Staubli VAL3: cycleStatus.pjx

--- cycleStatus.pjx ---
Parameters version=s7.5 stackSize=5000 millimeterUnit=true
Program file=addAction.pgx
Program file=addActionTime.pgx
Program file=addTraj.pgx
Program file=checkTollerance.pgx
Program file=getAction.pgx
Program file=getLastId.pgx
Program file=getSizeAction.pgx
Program file=getTraj.pgx
Program file=init.pgx
Program file=init_logAction.pgx
Program file=isActionEmpty.pgx
Program file=printLog.pgx
Program file=putInstr_Traj.pgx
Program file=recordPowerDown.pgx
Program file=removeAction.pgx
Program file=removeAllInstr.pgx
Program file=removeTraj.pgx
Data file=cycleStatus.dtx
Library alias=tcp path=Disk://kernel/tool/tool.pjx
Library alias=saveData path=Disk://saveData/saveData.pjx
Type name=TrajectoryItem path=Disk://kernel/template/TrajectoryItem/TrajectoryItem.pjx
Type name=ActionItem path=Disk://kernel/template/ActionItem/ActionItem.pjx
Type name=InstrItem path=Disk://kernel/template/InstrItem/InstrItem.pjx
Type name=progItem path=Disk://kernel/template/progItem/progItem.pjx
Type name=Trajectory path=Disk://kernel/template/Trajectory/Trajectory.pjx

--- cycleStatus.dtx ---
public ActionItem aActionTime
  [0]
    num nDistance = 1
    num nMoveId = 3
    num nTimeId
    num nPointId
    InstrItem iInstr[3]
      [0]
        string sType
        string sData
      [1]
        string sType
        string sData
      [2]
        string sType
        string sData
    string sIdTraj = "POINT place"
public InstrItem iToSuperV
  [0]
    string sType = "PROG"
    string sData = "home"
InstrItem tcpInstr[3]
  [0]
    string sType = "OUT"
    string sData = "bOut0>ON"
  [1]
    string sType = "OUT"
    string sData = "bOut1>OFF"
  [2]
    string sType
    string sData
Trajectory tTrajCycle
  [0]
    TrajectoryItem tSuper[3]
      [0]
        num distance
        num moveType = 1
        num nTime
        num nStop
        num nTcpAction
        string comment = "appro"
        bool toStop
        mdesc nom_speed = {tmax=1000, rmax=9999, leave=30, reach=30}
        InstrItem iInstr[3]
          [0]
            string sType
            string sData
          [1]
            string sType
            string sData
          [2]
            string sType
            string sData
        num nMoveId
      [1]
        num distance
        num moveType = 1
        num nTime
        num nStop
        num nTcpAction = 1
        string comment = "point"
        bool toStop = true
        mdesc nom_speed = {tmax=1000, rmax=9999, leave=30, reach=30}
        InstrItem iInstr[3]
          [0]
            string sType
            string sData
          [1]
            string sType
            string sData
          [2]
            string sType
            string sData
        num nMoveId
      [2]
        num distance
        num moveType = 1
        num nTime
        num nStop
        num nTcpAction
        string comment = "depart"
        bool toStop
        mdesc nom_speed = {tmax=1000, rmax=9999, leave=30, reach=30}
        InstrItem iInstr[3]
          [0]
            string sType
            string sData
          [1]
            string sType
            string sData
          [2]
            string sType
            string sData
        num nMoveId = 127
    string sID = "POINT pick"
    num nId
bool bActionMutex
public bool bAutoON
public bool bCALL
public bool bCycle
public bool bEnding
public bool bGOTO
public bool bHomeLoaded = true
public bool bHoming
public bool bIsHome
bool bLogMutex
public bool bMotionToken
public bool bMoveStopped
public bool bMutex
public bool bPause
public bool bPausePLC
public bool bShowMessage
public bool bSimulation
public bool bStop
public bool bToEnd
public bool bToHome
public bool bToPause
public bool bToStart
public bool bToStop
public bool bTrackEnable
public bool bTraj = true
public bool bWait
public bool bWritingToLog
public num nClockAction = 7230.098
public num nCycleTime = 1.833
public num nEmergency
public num nEvent
public num nIdPercentage = 5.617
public num nInterfaceToSV = -1
public num nLastIdPoint
public num nLastTimer = 5.715
public num nPoint = 2
public num nProcessType = 1
public num nProg
public num nTime = 7764.435
public num nToSuperV = -1
num nTollerance = 150
public num nWorkingMode = 4
public num nWorkingStatus = 2
pointRx pTollerance = {x=387.992409, y=64.919473, z=-164.968083, rx=0.107448, ry=178.01498, rz=42.225142, shoulder=lefty, elbow=epositive, wrist=wpositive, fatherId=world[0]}
public progItem pCycleProg
  [0]
    InstrItem iEvent[2]
      [0]
        string sType = "POINT"
        string sData = "pick"
      [1]
        string sType = "POINT"
        string sData = "place"
    string sID = "pick_place"
public string sLastAction = "OUT bOut0>OFF"
public string sToShow
public string sTraj
public string sTrajItem
ActionItem aActionTCP
  [0]
    num nDistance
    num nMoveId
    num nTimeId
    num nPointId
    InstrItem iInstr[3]
      [0]
        string sType
        string sData
      [1]
        string sType
        string sData
      [2]
        string sType
        string sData
    string sIdTraj
ActionItem aActionPoint
  [0]
    num nDistance
    num nMoveId
    num nTimeId
    num nPointId
    InstrItem iInstr[3]
      [0]
        string sType
        string sData
      [1]
        string sType
        string sData
      [2]
        string sType
        string sData
    string sIdTraj
public bool bActionRunning
ActionItem aAction
  [0]
    num nDistance
    num nMoveId
    num nTimeId
    num nPointId
    InstrItem iInstr[3]
      [0]
        string sType
        string sData
      [1]
        string sType
        string sData
      [2]
        string sType
        string sData
    string sIdTraj
public string sLog
public num nTimeMould[2]

--- addAction.pgx ---
public program addAction(ActionItem& x_aAction[])
  local num l_nSizeAction
  local num l_nSize
  local num l_nIndex
begin
  // mutex it
  setMutex(bActionMutex)
  //
  // insert a new action
  //
  if aAction.iInstr.sType!="null"
    append(aAction)
  endIf
  // set the size
  l_nSizeAction=size(aAction)-1
  // copy it
  aAction[l_nSizeAction]=x_aAction
  // update the nMoveId...
  l_nSize=size(tTrajCycle)-1
  l_nIndex=min(x_aAction.nPointId,size(tTrajCycle[l_nSize].tSuper)-1)
  tTrajCycle[l_nSize].tSuper[l_nIndex].nMoveId=x_aAction.nMoveId
  // release
  bActionMutex=false
end

--- addActionTime.pgx ---
public program addActionTime(ActionItem& x_aAction[] (dimensions=1))
  local num l_nSize[2]
begin
  // mutex
  setMutex(bLogMutex)
  // add one action with the timing
  if x_aAction.iInstr.sType==""
    // init
    aActionTime=x_aAction
  else
    // insert
    append(aActionTime)
    aActionTime[size(aActionTime)-1]=x_aAction
    aActionTime[size(aActionTime)-1].nTimeId=clock()-nClockAction
  endIf
  // update
  nClockAction=clock()
  //
  bLogMutex=false
end

--- addTraj.pgx ---
public program addTraj(Trajectory& x_tTrajectory)
  local num l_nSize
begin
  // mutex it
  setMutex(bActionMutex)
  if saveData:bDebug
    ? "TRAJ: Add "+x_tTrajectory.sID
  endIf
  //
  // insert a new action
  //
  if tTrajCycle.sID!="null" and tTrajCycle.sID!=""
    append(tTrajCycle)
  endIf
  // set the size
  l_nSize=size(tTrajCycle)-1
  // copy it
  tTrajCycle[l_nSize]=x_tTrajectory
  tTrajCycle[l_nSize].nId=nLastIdPoint
  // release
  bActionMutex=false
end

--- checkTollerance.pgx ---
public program checkTollerance(bool& x_bOk (dimensions=1))
begin
  if distance(here(flange,world),pTollerance)<nTollerance
    x_bOk=true
  else
    x_bOk=false
  endIf
end

--- getAction.pgx ---
public program getAction(ActionItem& x_aAction (dimensions=1))
begin
  // mutex it
  setMutex(bActionMutex)
  // give back the action on first element
  x_aAction=aAction[0]
  //release
  bActionMutex=false
end

--- getLastId.pgx ---
public program getLastId(num& x_nMoveId)
begin
  // give back the last ID
  x_nMoveId=aAction[size(aAction)-1].nMoveId
end

--- getSizeAction.pgx ---
public program getSizeAction(num& x_nSize)
begin
  // mutex it
  setMutex(bActionMutex)
  // give back the action on first element
  x_nSize=size(aAction)
  //release
  bActionMutex=false
end

--- getTraj.pgx ---
public program getTraj(Trajectory& x_tTrajectory (dimensions=1))
  local num l_nSize
begin
  // mutex it
  setMutex(bActionMutex)
  // get the first Traj
  x_tTrajectory=tTrajCycle[0]
  // release
  bActionMutex=false
end

--- init.pgx ---
public program init()
// initialization of the cycle
  local num i
  local num index
  local num hours
  local num l_nSize
begin
  // init all the cyclestatus variable
  //
  // BOOLEAN
  //
  // mutex
  bActionMutex=false
  bLogMutex=false
  // mutex it
  setMutex(bActionMutex)
  // use for pause the cycle
  bPause=false
  bToPause=false
  bPausePLC=false
  // use to goto another program and not came back
  bGOTO=false
  // use to call an other program and came back
  bCALL=false
  // use to wait after an input
  bWait=false
  // init the restart MOVE
  bMoveStopped=false
  // set the motion token to false
  bMotionToken=false
  // use to see if is going to home
  bHoming=false
  // show a message on the screen
  bShowMessage=false
  // auto_on
  bAutoON=false
  // stop motion control
  bStop=false
  // the stop boolean
  bToStop=false
  // use to end the cycle
  bToEnd=false
  bEnding=false
  // to start the cycle
  bToStart=false
  // to homing
  bToHome=false
  bHoming=false
  // reset TASK CONTROL
  bActionRunning=false
  // STRING
  //
  // show the event that is processing
  sToShow=""
  //
  // INTEGER
  //
  // cycleEvent
  nEvent=0
  nPoint=0
  nProg=0
  // cycle Type
  nProcessType=0
  // ACTION
  resize(aAction,1,1)
  resize(aAction.iInstr,1,3)
  aAction.iInstr.sType="null"
  aAction.iInstr.sData=""
  aAction.iInstr[1].sType="null"
  aAction.iInstr[1].sData=""
  aAction.iInstr[2].sType="null"
  aAction.iInstr[2].sData=""
  aAction.nMoveId=-1
  aAction.nPointId=0
  aAction.sIdTraj="null"
  // TRAJECTORY
  resize(tTrajCycle,1,1)
  tTrajCycle.sID="null"
  resize(tTrajCycle.tSuper,1,1)
  // PROGRAM
  resize(pCycleProg.iEvent,1,1)
  pCycleProg.iEvent.sType=""
  pCycleProg.iEvent.sData=""
  pCycleProg.sID=""
  // release
  bActionMutex=false
end

--- init_logAction.pgx ---
public program init_logAction()
  local num l_nSize
  local num i
begin
  // mutex it
  setMutex(bLogMutex)
  // logAction
  resize(sLog,1,1)
  sLog=""
  bLogMutex=false
end

--- isActionEmpty.pgx ---
public program isActionEmpty(bool& x_bEmpty)
begin
  // check if there are some action in the queue
  if aAction.iInstr.sType!="null"
    x_bEmpty=false
  else
    x_bEmpty=true
  endIf
end

--- printLog.pgx ---
public program printLog(string x_sMessage)
  local num i
  local num l_nSize
begin
  // check the size after is 200 clear it and keep the first 50
  setMutex(bLogMutex)
  // do it
  if size(sLog)>=200
    // clean it
    delete(sLog[0])
  endIf
  // add one
  if sLog!=""
    insert(sLog[size(sLog)])
  endIf
  // write it
  sLog[size(sLog)-1]=x_sMessage
  //release
  bLogMutex=false
end

--- putInstr_Traj.pgx ---
public program putInstr_Traj(ActionItem& x_aAction[], TrajectoryItem x_tTrajItem, num x_nTCP, num x_nSize)
  local num j
  local tool l_tTool
begin
  // save the data
  aActionTCP.nMoveId=aActionPoint.nMoveId=x_aAction.nMoveId
  aActionTCP.nPointId=aActionPoint.nPointId=x_aAction.nPointId
  // use the blend anticipation for the last point
  if aActionPoint.nPointId==x_nSize-1 and x_tTrajItem.nom_speed.blend!=off and saveData:bUseBlendAction
    x_tTrajItem.distance=max(x_tTrajItem.distance,x_tTrajItem.nom_speed.leave+5)
  endIf
  aActionPoint.nDistance=(max(100-(x_tTrajItem.distance*100/max(x_aAction.nDistance,1)),0))/100
  aActionTCP.nTimeId=aActionPoint.nTimeId=x_aAction.nTimeId
  aActionTCP.sIdTraj=aActionPoint.sIdTraj=x_aAction.sIdTraj
  // ADD the instruction
  // TCP ON OFF
  if x_tTrajItem.nTcpAction>0
    // get the instruction items
    call tcp:getInstr(aActionTCP.iInstr,x_tTrajItem.nTcpAction==1,x_nTCP)
    // get the time delay
    call tcp:getTool(l_tTool,x_nTCP)
    switch x_tTrajItem.nTcpAction
      case 1
        aActionTCP.nDistance=l_tTool.otime
      break
      case 2
        aActionTCP.nDistance=l_tTool.ctime
      break
    endSwitch
    if aActionTCP.nPointId==x_nSize-1 and x_tTrajItem.nom_speed.blend!=off and saveData:bUseBlendAction
      aActionTCP.nDistance=max(aActionTCP.nDistance,x_tTrajItem.nom_speed.leave+5)
    endIf
    // use the blend anticipation for the last point
    aActionTCP.nDistance=(max(100-(aActionTCP.nDistance*100/max(x_aAction.nDistance,1)),0))/100
    // insert in the stack
    call addAction(aActionTCP)
  endIf
  // ON POINT
  for j=0 to size(x_tTrajItem.iInstr)-1
    aActionPoint.iInstr[j]=x_tTrajItem.iInstr[j]
  endFor
  // insert in the stack
  call addAction(aActionPoint)
end

--- recordPowerDown.pgx ---
public program recordPowerDown()
begin
  // record the powerDown point
  pTollerance=here(flange,world)
end

--- removeAction.pgx ---
public program removeAction()
begin
  // mutex it
  setMutex(bActionMutex)
  // remove the action
  if size(aAction)>1
    delete(aAction[0])
  else
    // remove
    resize(aAction[0].iInstr,1,1)
    aAction[0].iInstr.sType="null"
    aAction[0].iInstr.sData=""
    aAction.nPointId=0
  endIf
  // release
  bActionMutex=false
end

--- removeAllInstr.pgx ---
public program removeAllInstr(ActionItem& x_aAction[], TrajectoryItem x_tTrajItem, num x_nTCP, num x_nSize)
  local num j
  local tool l_tTool
begin
  // save the data
  aActionTCP.nMoveId=aActionPoint.nMoveId=x_aAction.nMoveId
  aActionTCP.nPointId=aActionPoint.nPointId=x_aAction.nPointId
  // use the blend anticipation for the last point
  if aActionPoint.nPointId==x_nSize-1 and x_tTrajItem.nom_speed.blend!=off and saveData:bUseBlendAction
    x_tTrajItem.distance=max(x_tTrajItem.distance,x_tTrajItem.nom_speed.leave+5)
  endIf
  aActionPoint.nDistance=(max(100-(x_tTrajItem.distance*100/max(x_aAction.nDistance,1)),0))/100
  aActionTCP.nTimeId=aActionPoint.nTimeId=x_aAction.nTimeId
  aActionTCP.sIdTraj=aActionPoint.sIdTraj=x_aAction.sIdTraj
  // ADD the instruction
  // TCP ON OFF
  if x_tTrajItem.nTcpAction>0
    // get the instruction items
    call tcp:getInstr(aActionTCP.iInstr,x_tTrajItem.nTcpAction==1,x_nTCP)
    // get the time delay
    call tcp:getTool(l_tTool,x_nTCP)
    switch x_tTrajItem.nTcpAction
      case 1
        aActionTCP.nDistance=l_tTool.otime
      break
      case 2
        aActionTCP.nDistance=l_tTool.ctime
      break
    endSwitch
    if aActionTCP.nPointId==x_nSize-1 and x_tTrajItem.nom_speed.blend!=off and saveData:bUseBlendAction
      aActionTCP.nDistance=max(aActionTCP.nDistance,x_tTrajItem.nom_speed.leave+5)
    endIf
    // use the blend anticipation for the last point
    aActionTCP.nDistance=(max(100-(aActionTCP.nDistance*100/max(x_aAction.nDistance,1)),0))/100
    // insert in the stack
    call addAction(aActionTCP)
  endIf
  // ON POINT
  for j=0 to size(x_tTrajItem.iInstr)-1
    aActionPoint.iInstr[j]=x_tTrajItem.iInstr[j]
  endFor
  // insert in the stack
  call addAction(aActionPoint)
end

--- removeTraj.pgx ---
public program removeTraj()
begin
  // mutex it
  setMutex(bActionMutex)
  if saveData:bDebug
    ? "CYCLESTATUS: TRAJ Remove "+tTrajCycle.sID
  endIf
  // remove the action
  if size(tTrajCycle)>1
    delete(tTrajCycle[0])
  else
    // reset
    resize(tTrajCycle.tSuper,1,1)
    tTrajCycle.sID="null"
    tTrajCycle.nId=0
  endIf
  // release
  bActionMutex=false
end
